FUNCTION_BLOCK FB_CheckOperation
VAR
	
	StartTimer : TON;
	TimerDone : BOOL;
	
	Counter : CTU; 
	ResetCommand : BOOL; 
END_VAR

StartTimer(IN:= GVL.OperationStart , PT:= T#2S);
TimerDone := StartTimer.Q; 

IF TimerDone THEN  
	gvl.LoadMeasurementStart := TRUE;
ELSE
	gvl.LoadMeasurementWait := TRUE;
END_IF

//Counter(
	//CU:=TimerDone , 
	//RESET:= ResetCommand , 
	//PV:= 5);

END_FUNCTION_BLOCK

(* stored: Version 1.1.0.1, ProductVersion 3.1.4024.12
   POU FB_CheckOperation: Id {8705b537-706d-4801-b262-e6d5a3b0b4d3}, SpecialFunc None *)
